{attribute 'no_explicit_call' := 'do not call this function block directly'}
{attribute 'OPC.UA.DA' := '0'}
FUNCTION_BLOCK INTERNAL UnifiedProgramStepExecutor EXTENDS ToolkitObject
VAR_STAT
	//! <summary>Class name shared by all instances of this function block.</summary>
	_ClassName : STRING := __POUNAME();
END_VAR
VAR
	_StateMachine : REFERENCE TO UnifiedProgramStateMachine;
	
	_ExecutedSteps : ARRAY [0..UnifiedProgramConstants.MaxStepCount - 1] OF UNIFIED_PROGRAM_EXECUTED_STEP;
	_ExecutedStepCount : INT;
	_ExecutedStep : REFERENCE TO UNIFIED_PROGRAM_EXECUTED_STEP;	
END_VAR

{attribute 'monitoring' := 'call'}
PROPERTY ClassName : REFERENCE TO STRING
GET
ClassName REF= _ClassName;
END_GET
END_PROPERTY

METHOD FB_init : BOOL
VAR_INPUT
	bInitRetains : BOOL; // TRUE: the retain variables are initialized (reset warm / reset cold)
	bInCopyCode : BOOL;  // TRUE: the instance will be copied to the copy code afterward (online change)
	stateMachine : REFERENCE TO UnifiedProgramStateMachine;
END_VAR
_StateMachine REF= stateMachine;
END_METHOD

METHOD Reset 
VAR
	i : DINT;
END_VAR
FOR i := 0 TO UnifiedProgramConstants.MaxStepCount - 1 DO
	_ExecutedSteps[i].StepIndex := -1;
	_ExecutedSteps[i].Step REF= 0;
END_FOR

_ExecutedStepCount := 0;
_ExecutedStep REF= 0;
END_METHOD

END_FUNCTION_BLOCK

(* stored: Version 1.1.0.1
   POU UnifiedProgramStepExecutor: Id {6e5659b6-0a9c-47f4-b9aa-f36926b112ec}, SpecialFunc None
   Property ClassName: Id {c6657840-2637-41bc-bc1f-a8a05273ac50}
   Get Get: Id {ee552158-e6d5-4e6e-aceb-9ce9c5786526}
   Method FB_init: Id {bed5f855-ec00-4e82-b315-2ade88b8b0ee}
   Method Reset: Id {b699b8ec-3ffc-44f1-9c96-795957b17c22} *)
